RoboDK station: Bir-main_alter_newtool.rdk

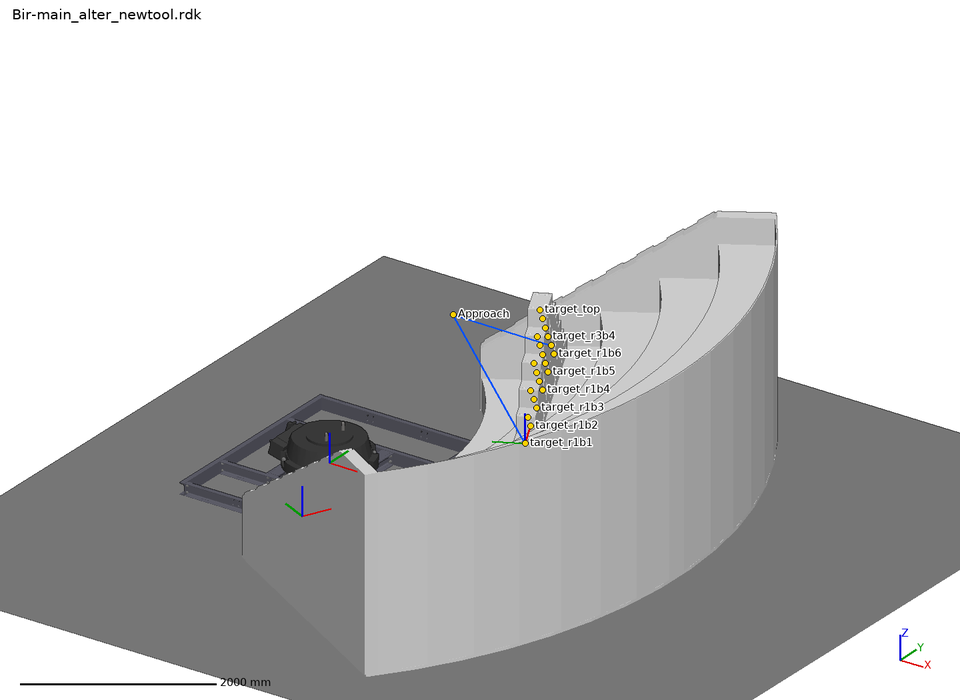
[picture v0: the station drawn from its stored meshes, robots at their saved joint values, targets as dots, program paths as lines]
Station Bir-main_alter_newtool (saved by RoboDK 5.4.1). Poses are relative to the parent item; angles as X-Y-Z fixed-axis rotations.
  - folder assets
    - object Floor at (0, 0, 0) mm, size 9000 x 9000 x 0 mm, geometry from Floor.sld
    - object Stairs_v1 at (-2520, 0, 0) mm, size 3922.2 x 7408.9 x 2302 mm, geometry from Stairs_v1.3ds
    - object Frame at (0, 0, 0) mm, size 2000 x 2500 x 199.8 mm, geometry from Frame.stp
  - frame KUKA KR 210-2 Base at (0, 0, 140) mm
    - robot KUKA KR 210-2: 6 axes, payload 210 kg, reach 2700 mm, repeatability 0.06 mm, weight 1267 kg
        joint limits [-185, -146, -119, -350, -125, -350] to [185, 0, 155, 350, 125, 350]; home [0, -90, 90, 0, 0, 0]; saved at [65.098, -124.848, 131.589, -277.937, -40.566, 280.4]
      - tool NEMO_ASM-v2, TCP at (50, 0, 430) mm, size 350 x 350 x 427.5 mm, geometry from NEMO_ASM-v2.stp
    - frame Table 1 at (2270, 238.94, 760) mm, rotated rx 0 ry 0 rz 117 deg
      - target Approach (Cartesian target) at (1070, 893.91, 882.09) mm, rotated rx 0 ry 90 rz -90 deg; joints [-50.616, -131.085, 128.227, -276.506, 23.778, 277.104] of KUKA KR 210-2
      - target target_top (Cartesian target) at (1070, 0, 1000) mm, rotated rx 0 ry 90 rz -90 deg; joints [-36.734, -87.365, 94.367, -234.601, 11.971, 234.004] of KUKA KR 210-2
      - target target_r1b1 (Cartesian target) at (0, 0, 0) mm, rotated rx 0 ry 90 rz -90 deg; joints [2.067, -52.896, 108.321, -145.978, 60.263, 161.487] of KUKA KR 210-2
      - target target_r1b2 (Cartesian target) at (420, 0, 0) mm, rotated rx 0 ry 90 rz -90 deg; joints [-11.873, -56.834, 117.553, -162.781, 61.827, 171.675] of KUKA KR 210-2
      - target target_r1b3 (Cartesian target) at (840, 0, 0) mm, rotated rx 0 ry 90 rz -90 deg; joints [-27.87, -58.059, 120.514, -180.981, 62.458, 180.454] of KUKA KR 210-2
      - target target_r1b4 (Cartesian target) at (1260, 0, 0) mm, rotated rx 0 ry 90 rz -90 deg; joints [-43.736, -56.543, 116.857, -199.092, 61.689, 189.322] of KUKA KR 210-2
      - target target_r1b5 (Cartesian target) at (1680, 0, 0) mm, rotated rx 0 ry 90 rz -90 deg; joints [-57.379, -52.32, 106.997, -215.696, 60.08, 199.716] of KUKA KR 210-2
      - target target_r1b6 (Cartesian target) at (2100, 0, 0) mm, rotated rx 0 ry 90 rz -90 deg; joints [-68.079, -45.403, 91.45, -230.448, 58.454, 212.354] of KUKA KR 210-2
      - target target_r2b1 (Cartesian target) at (210, 0, 200) mm, rotated rx 0 ry 90 rz -90 deg; joints [-4.556, -63.685, 112.198, -151.127, 52.247, 161.345] of KUKA KR 210-2
      - target target_r2b2 (Cartesian target) at (630, 0, 200) mm, rotated rx 0 ry 90 rz -90 deg; joints [-19.73, -67.105, 118.287, -170.702, 51.551, 174.187] of KUKA KR 210-2
      - target target_r2b3 (Cartesian target) at (1050, 0, 200) mm, rotated rx 0 ry 90 rz -90 deg; joints [-35.975, -66.907, 117.939, -191.483, 51.597, 187.192] of KUKA KR 210-2
      - target target_r2b4 (Cartesian target) at (1470, 0, 200) mm, rotated rx 0 ry 90 rz -90 deg; joints [-50.915, -63.129, 111.192, -210.8, 52.343, 200.011] of KUKA KR 210-2
      - target target_r2b5 (Cartesian target) at (1890, 0, 200) mm, rotated rx 0 ry 90 rz -90 deg; joints [-63.09, -56.325, 98.57, -227.315, 53.258, 212.968] of KUKA KR 210-2
      - target target_r3b1 (Cartesian target) at (420, 0, 400) mm, rotated rx 0 ry 90 rz -90 deg; joints [-11.873, -73.433, 112.651, -156.851, 41.591, 162.268] of KUKA KR 210-2
      - target target_r3b2 (Cartesian target) at (840, 0, 400) mm, rotated rx 0 ry 90 rz -90 deg; joints [-27.87, -75.428, 115.47, -181.352, 40.05, 181.035] of KUKA KR 210-2
      - target target_r3b3 (Cartesian target) at (1260, 0, 400) mm, rotated rx 0 ry 90 rz -90 deg; joints [-43.736, -72.971, 111.985, -205.532, 41.92, 199.566] of KUKA KR 210-2
      - target target_r3b4 (Cartesian target) at (1680, 0, 400) mm, rotated rx 0 ry 90 rz -90 deg; joints [-57.379, -66.672, 102.456, -225.072, 45.585, 215.054] of KUKA KR 210-2
      - target target_r4b1 (Cartesian target) at (640, 0, 600) mm, rotated rx 0 ry 90 rz -90 deg; joints [-20.114, -81.144, 109.759, -165.847, 29.364, 167.605] of KUKA KR 210-2
      - target target_r4b2 (Cartesian target) at (1060, 0, 600) mm, rotated rx 0 ry 90 rz -90 deg; joints [-36.355, -80.757, 109.291, -199.028, 29.906, 196.644] of KUKA KR 210-2
      - target target_r4b3 (Cartesian target) at (1480, 0, 600) mm, rotated rx 0 ry 90 rz -90 deg; joints [-51.24, -75.656, 102.814, -224.608, 35.776, 218.67] of KUKA KR 210-2
      - target target_r5b1 (Cartesian target) at (860, 0, 800) mm, rotated rx 0 ry 90 rz -90 deg; joints [-28.649, -85.852, 103.546, -185.41, 17.768, 185.153] of KUKA KR 210-2
      - target target_r5b2 (Cartesian target) at (1280, 0, 800) mm, rotated rx 0 ry 90 rz -90 deg; joints [-44.447, -82.727, 100.045, -226.556, 24.391, 223.879] of KUKA KR 210-2
      - object top_brick at (1070, 0, 1000) mm, size 400 x 200 x 210 mm, geometry from brick_Origin.sld
      - object row1brick1 at (0, 0, 0) mm, size 400 x 200 x 210 mm, geometry from brick_Origin.sld
        - object row1brick2 at (420, 0, 0) mm, size 400 x 200 x 210 mm, geometry from brick_Origin.sld
          - object row1brick3 at (420, 0, 0) mm, size 400 x 200 x 210 mm, geometry from brick_Origin.sld
            - object row1brick4 at (420, 0, 0) mm, size 400 x 200 x 210 mm, geometry from brick_Origin.sld
              - object row1brick5 at (420, 0, 0) mm, size 400 x 200 x 210 mm, geometry from brick_Origin.sld
                - object row1brick6 at (420, 0, 0) mm, size 400 x 200 x 210 mm, geometry from brick_Origin.sld
      - object row2brick1 at (210, 0, 200) mm, size 400 x 200 x 210 mm, geometry from brick_Origin.sld
        - object row2brick2 at (420, 0, 0) mm, size 400 x 200 x 210 mm, geometry from brick_Origin.sld
          - object row2brick3 at (420, 0, 0) mm, size 400 x 200 x 210 mm, geometry from brick_Origin.sld
            - object row2brick4 at (420, 0, 0) mm, size 400 x 200 x 210 mm, geometry from brick_Origin.sld
              - object row2brick5 at (420, 0, 0) mm, size 400 x 200 x 210 mm, geometry from brick_Origin.sld
      - object row3brick1 at (420, 0, 400) mm, size 400 x 200 x 210 mm, geometry from brick_Origin.sld
        - object row3brick2 at (420, 0, 0) mm, size 400 x 200 x 210 mm, geometry from brick_Origin.sld
          - object row3brick3 at (420, 0, 0) mm, size 400 x 200 x 210 mm, geometry from brick_Origin.sld
            - object row3brick4 at (420, 0, 0) mm, size 400 x 200 x 210 mm, geometry from brick_Origin.sld
      - object row4brick1 at (640, 0, 600) mm, size 400 x 200 x 210 mm, geometry from brick_Origin.sld
        - object row4brick2 at (420, 0, 0) mm, size 400 x 200 x 210 mm, geometry from brick_Origin.sld
          - object row4brick3 at (420, 0, 0) mm, size 400 x 200 x 210 mm, geometry from brick_Origin.sld
      - object row5brick1 at (860, 0, 800) mm, size 400 x 200 x 210 mm, geometry from brick_Origin.sld
        - object top_brick at (420, 0, 0) mm, size 400 x 200 x 210 mm, geometry from brick_Origin.sld
    - frame Table 2 at (1260, -2281.06, 660) mm, rotated rx 0 ry 0 rz 65 deg
      - target Target 1 (Cartesian target) at (3874.34, 1638.97, 300) mm, rotated rx 0 ry 90 rz -38 deg; joints [-115.064, -27.533, 36.078, -258.468, 36.928, 255.682] of KUKA KR 210-2
  - program Pick and place (13 instructions, listed below)
  - program Replace objects (1 instructions, listed below)
  - object brick at (-300, 3000, 0) mm, size 400 x 200 x 210 mm, geometry from brick.stp
  - object brick4 at (101.67, -1.69, 95.08) mm, size 400 x 200 x 210 mm, geometry from brick_Origin.sld
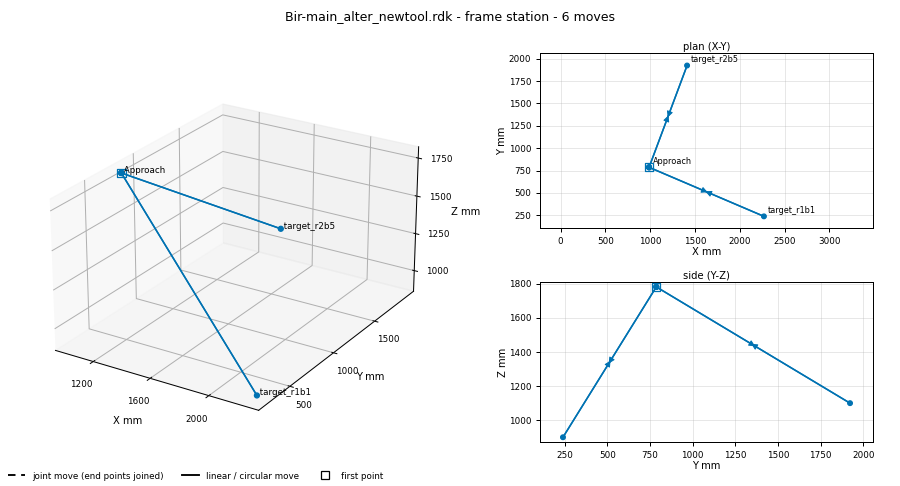
[picture p0: tool path of Bir-main_alter_newtool.rdk in frame station, 6 of 6 moves have a stored position in this frame; points joined in program order, loops and branches not executed]

--- program Pick and place (robot KUKA KR 210-2) ---
  Set Frame: Table 1
  Set Tool: NEMO_ASM-v2
  MoveJ (Approach)
  MoveL (target_top) -> target target_r2b5
  Attach to Tool
  Call AirValve_On
  MoveL (Approach)
  Set Ref.: Table 2
  MoveJ (Approach)
  MoveL (target_r1b1)
  Detach from Tool
  Call AirValve_Off
  MoveL (Approach)

--- program Replace objects (robot KUKA KR 210-2) ---
  Replace objects
